(* IEC 61131-3 sources: ae-debugging/src/classProgram, 1 file *)

(* ---- classProgram.st ---- *)
PROGRAM ClassProgram
    VAR_EXTERNAL
        GlobalInt : INT;
    END_VAR

    VAR
        localConveyorClass : Conveyor;
    END_VAR

    IF NOT localConveyorClass.is_running THEN
        localConveyorClass.Start();
    ELSE
        localConveyorClass.Stop();
    END_IF;

END_PROGRAM
